TEXTLIST EL1904_M_5
  1 = 'Safety output feedback 1' | chinese: '安全输出反馈1' | Chinese: '安全输出反馈1'
  2 = 'Safety output feedback 2' | chinese: '安全输出反馈2' | Chinese: '安全输出反馈2'
  3 = 'Safety output feedback 3' | chinese: '安全输出反馈3' | Chinese: '安全输出反馈3'
  4 = 'Safety output feedback 4' | chinese: '安全输出反馈4' | Chinese: '安全输出反馈4'
   = ''
END_TEXTLIST

(* stored: Version 1.1.0.1, ProductVersion 3.1.4024.11
   TextList EL1904_M_5: Id {6c6431a0-e255-455d-956e-5de7cbf4351c} *)
